# EPICS autosave request: apps/chillerApp/Db/Lauda_XT_settings.req
#
# Lauda Integral XT 150 Chiller
#
$(P)$(R)cooling_mode:set
$(P)$(R)outflow_temp:set
$(P)$(R)outflow_temp_lim_hi:set
$(P)$(R)outflow_temp_lim_low:set
